// Mitsubishi GX Works2 project: excercicio1   PLC: Q03UDV

PROGRAM MAIN
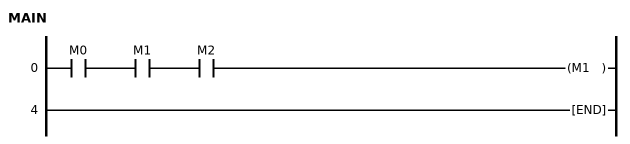
0     LD      M0
      AND     M1
      AND     M2
      OUT     M1
4     END
END_PROGRAM
